// Mitsubishi GX Works2 project: Test random   PLC: FX1N/FX1NC
// FX3S_Terco_Awal

PROGRAM MAIN  // ladder awal
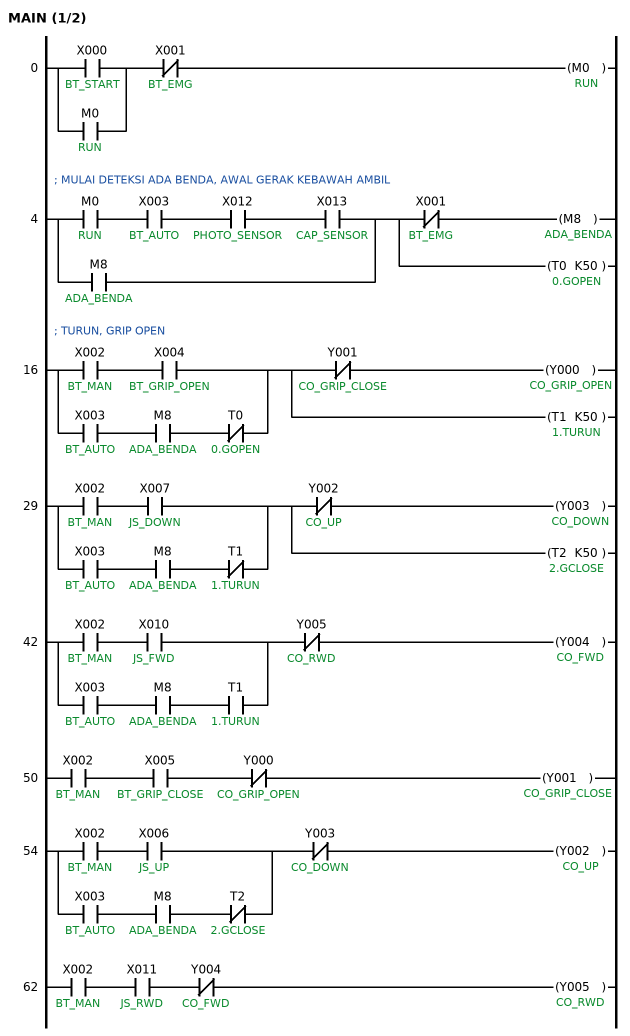
0     LD      X000  ; BT_START
      OR      M0  ; RUN
      ANI     X001  ; BT_EMG
      OUT     M0  ; RUN
; MULAI DETEKSI ADA BENDA, AWAL GERAK KEBAWAH AMBIL
4     LD      M0  ; RUN
      AND     X003  ; BT_AUTO
      AND     X012  ; PHOTO_SENSOR
      AND     X013  ; CAP_SENSOR
      OR      M8  ; ADA_BENDA
      MPS
      ANI     X001  ; BT_EMG
      OUT     M8  ; ADA_BENDA
      MPP
      OUT     T0 K50  ; 0.GOPEN
; TURUN, GRIP OPEN
16    LD      X002  ; BT_MAN
      AND     X004  ; BT_GRIP_OPEN
      LD      X003  ; BT_AUTO
      AND     M8  ; ADA_BENDA
      ANI     T0  ; 0.GOPEN
      ORB
      MPS
      ANI     Y001  ; CO_GRIP_CLOSE
      OUT     Y000  ; CO_GRIP_OPEN
      MPP
      OUT     T1 K50  ; 1.TURUN
29    LD      X002  ; BT_MAN
      AND     X007  ; JS_DOWN
      LD      X003  ; BT_AUTO
      AND     M8  ; ADA_BENDA
      ANI     T1  ; 1.TURUN
      ORB
      MPS
      ANI     Y002  ; CO_UP
      OUT     Y003  ; CO_DOWN
      MPP
      OUT     T2 K50  ; 2.GCLOSE
42    LD      X002  ; BT_MAN
      AND     X010  ; JS_FWD
      LD      X003  ; BT_AUTO
      AND     M8  ; ADA_BENDA
      AND     T1  ; 1.TURUN
      ORB
      ANI     Y005  ; CO_RWD
      OUT     Y004  ; CO_FWD
50    LD      X002  ; BT_MAN
      AND     X005  ; BT_GRIP_CLOSE
      ANI     Y000  ; CO_GRIP_OPEN
      OUT     Y001  ; CO_GRIP_CLOSE
54    LD      X002  ; BT_MAN
      AND     X006  ; JS_UP
      LD      X003  ; BT_AUTO
      AND     M8  ; ADA_BENDA
      ANI     T2  ; 2.GCLOSE
      ORB
      ANI     Y003  ; CO_DOWN
      OUT     Y002  ; CO_UP
62    LD      X002  ; BT_MAN
      AND     X011  ; JS_RWD
      ANI     Y004  ; CO_FWD
      OUT     Y005  ; CO_RWD
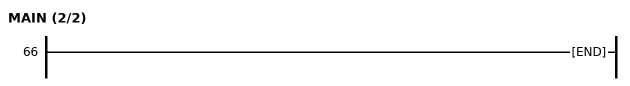
66    END
END_PROGRAM

// device comments not shown above
M1  ; GOPEN_MAN
M2  ; GCLOSE_MAN
M3  ; UP_MAN
M4  ; DOWN_MAN
M5  ; FWD_MAN
M6  ; RWD_MAN
M7  ; MODERESET
M100  ; Fl_tangan
M101  ; Fl_posY
M102  ; Fl_posX
